// LS Electric XG5000 project: 동남113
// PLC NewPLC
// module base 0 slot 0: 입출력 모듈:XBC-DN/DP14E (DC 24V 입력 8점, 트랜지스터 출력 6점)

PROGRAM NewProgram (task: 스캔 프로그램)

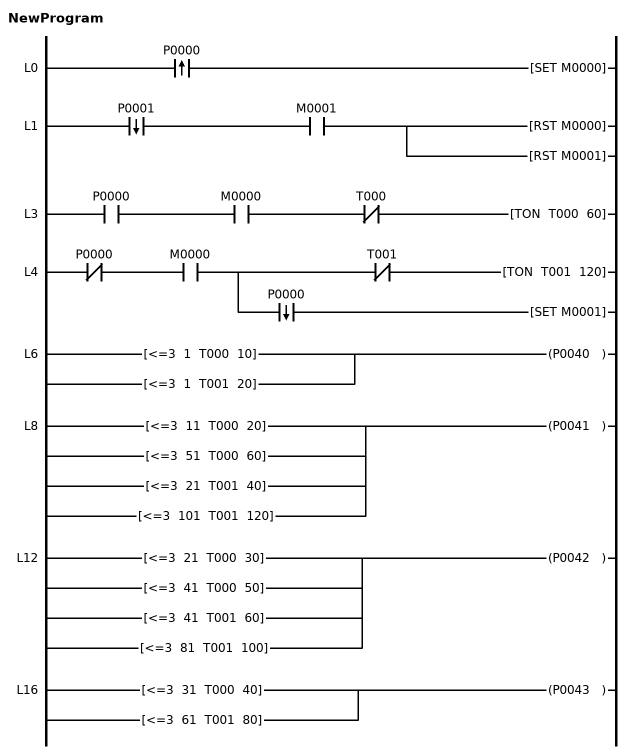
; L0
LOADP     P0000
SET       M0000
; L1
LOADN     P0001
AND       M0001
RST       M0000
RST       M0001
; L3
LOAD      P0000
AND       M0000
AND NOT   T000
TON       T000 60
; L4
LOAD NOT  P0000
AND       M0000
MPUSH
AND NOT   T001
TON       T001 120
MPOP
ANDN      P0000
SET       M0001
; L6
LOAD<=3   1 T000 10
OR<=3     1 T001 20
OUT       P0040
; L8
LOAD<=3   11 T000 20
OR<=3     51 T000 60
OR<=3     21 T001 40
OR<=3     101 T001 120
OUT       P0041
; L12
LOAD<=3   21 T000 30
OR<=3     41 T000 50
OR<=3     41 T001 60
OR<=3     81 T001 100
OUT       P0042
; L16
LOAD<=3   31 T000 40
OR<=3     61 T001 80
OUT       P0043